// TIA Portal V20 export
// export: Created 2025-12-01T14:57:30.722672Z, ExportSetting None, DisplayName Totally Integrated Automation Portal, DisplayVersion V20 Update 3, DisplayName TIA Portal Openness, DisplayVersion V20 Update 3, DisplayName TIA Portal Version Control Interface, DisplayVersion V20 Update 3, DisplayName STEP 7 Professional, DisplayVersion V20 Update 3, DisplayName STEP 7 Safety, DisplayVersion V20 Update 2, DisplayName WinCC Basic/Comfort/Advanced, DisplayVersion V20 Update 3, DisplayName WinCC Professional, DisplayVersion V20 Update 3, DisplayName WinCC Unified, DisplayVersion V20 Update 3
FUNCTION_BLOCK "FB1700_Activacion_tarjetas"   // FB1700, LAD
{ S7_Optimized_Access := 'TRUE' }
// Este bloque cambiara la variable de salida entre 1 y 5, este cambio se realizara despues de un tiempo.
// stored: AutoNumber false, MemoryReserve 100, SetENOAutomatically false
   VAR_INPUT
      v_Tiempo_por_posicion : Time;
   END_VAR
   VAR_OUTPUT
      Num_de_posicion_en_la_linea : Byte;
   END_VAR
   VAR DB_SPECIFIC
      Mx_ET00 : Bool;
      Mx_ET01 : Bool;
      Mx_ET02 : Bool;
      Mx_ET03 : Bool;
   END_VAR
   VAR
      Tiempo_por_posicion : TON_TIME;
      Posicion { S7_SetPoint := 'True'} : Byte;
      FP_Contador : Bool;
   END_VAR
BEGIN

REGION Network 2: ET01 - ESTADO REPOSO VACIO
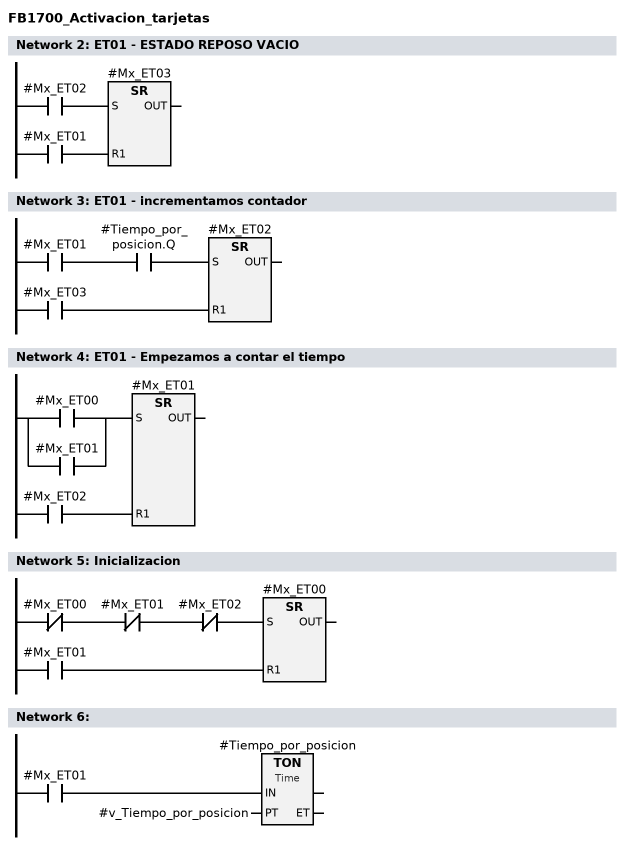
   RUNG wire#powerrail
      Contact( #Mx_ET02 )
      S_SR(operand := #Mx_ET03, r1 := wire#w1)
   END_RUNG
   RUNG wire#powerrail
      Contact( #Mx_ET01 )
   END_RUNG wire#w1
   // the same network as SCL:
   IF #Mx_ET02 THEN
       #Mx_ET03 := TRUE;   // SR flip-flop
   END_IF;
   IF #Mx_ET01 THEN #Mx_ET03 := FALSE; END_IF;
END_REGION

REGION Network 3: ET01 - incrementamos contador
   RUNG wire#powerrail
      Contact( #Mx_ET01 )
      Contact( #Tiempo_por_posicion.Q )
      S_SR(operand := #Mx_ET02, r1 := wire#w1)
   END_RUNG
   RUNG wire#powerrail
      Contact( #Mx_ET03 )
   END_RUNG wire#w1
   // the same network as SCL:
   IF #Mx_ET01 AND #Tiempo_por_posicion.Q THEN
       #Mx_ET02 := TRUE;   // SR flip-flop
   END_IF;
   IF #Mx_ET03 THEN #Mx_ET02 := FALSE; END_IF;
END_REGION

REGION Network 4: ET01 - Empezamos a contar el tiempo
   RUNG wire#powerrail
      Contact( #Mx_ET00 )
      wire#w1
      S_SR(operand := #Mx_ET01, r1 := wire#w2)
   END_RUNG
   RUNG wire#powerrail
      Contact( #Mx_ET01 )
   END_RUNG wire#w1
   RUNG wire#powerrail
      Contact( #Mx_ET02 )
   END_RUNG wire#w2
   // the same network as SCL:
   IF #Mx_ET00 OR #Mx_ET01 THEN
       #Mx_ET01 := TRUE;   // SR flip-flop
   END_IF;
   IF #Mx_ET02 THEN #Mx_ET01 := FALSE; END_IF;
END_REGION

REGION Network 5: Inicializacion
   RUNG wire#powerrail
      I_Contact( #Mx_ET00 )
      I_Contact( #Mx_ET01 )
      I_Contact( #Mx_ET02 )
      S_SR(operand := #Mx_ET00, r1 := wire#w1)
   END_RUNG
   RUNG wire#powerrail
      Contact( #Mx_ET01 )
   END_RUNG wire#w1
   // the same network as SCL:
   IF NOT #Mx_ET00 AND NOT #Mx_ET01 AND NOT #Mx_ET02 THEN
       #Mx_ET00 := TRUE;   // SR flip-flop
   END_IF;
   IF #Mx_ET01 THEN #Mx_ET00 := FALSE; END_IF;
END_REGION

REGION Network 6
   RUNG wire#powerrail
      Contact( #Mx_ET01 )
      { S7_Templates := "time_type := Time" } #Tiempo_por_posicion.TON(pt := #v_Tiempo_por_posicion, et =>)
   END_RUNG
   // the same network as SCL:
   #Tiempo_por_posicion(IN := #Mx_ET01, PT := #v_Tiempo_por_posicion);   // TON
END_REGION

NETWORK
TITLE = Incrementamos el contador
//en la etapa 1 incrementamos el contador
      A     #Mx_ET01;
      FP    #FP_Contador;
      JCN   salto;

      L     1;
      L     #Posicion;
      +I;
      T     #Posicion;


//si una vez que incrementamos el contador, el contador es mayor a 5 entonces volvemos a empezar
      L     #Posicion;
      L     5;
      <=I;
      JC    iniciar;

      L     1;
      T     #Posicion;

iniciar:NOP   0;



salto:NOP   0;


      L     #Posicion;
      T     #Num_de_posicion_en_la_linea;



END_FUNCTION_BLOCK
